// TIA Portal V21 export
DATA_BLOCK "DB_Celda"   // DB1
{ S7_Optimized_Access := 'TRUE' }
// stored: MemoryReserve 100
   VAR
      Caja : "UDT_ Caja";
      Contador { S7_SetPoint := 'True'} : "UDT_Contador";
      "Sistema en marcha" { S7_SetPoint := 'True'} : Bool;
      "Modo auto" { S7_SetPoint := 'True'} : Bool;
      Emergencia { S7_SetPoint := 'True'} : Bool;
      Clasificando { S7_SetPoint := 'True'} : Bool;
   END_VAR
BEGIN
END_DATA_BLOCK
